{attribute 'no_explicit_call':= 'do not call this POU directly'}
FUNCTION_BLOCK TValueMonitor
VAR
    _CurrentValue : INT := -1;
    _PreviousValue : INT;
    _Changed : BOOL;
END_VAR

PROPERTY Changed : BOOL
GET
Changed := _Changed;
END_GET
END_PROPERTY

PROPERTY CurrentValue : INT
GET
CurrentValue := _CurrentValue;
END_GET
END_PROPERTY

PROPERTY PreviousValue : INT
GET
PreviousValue := _PreviousValue;
END_GET
END_PROPERTY

METHOD Reset
VAR_INPUT
END_VAR
_CurrentValue := 0;
_PreviousValue := 0;
END_METHOD

METHOD Test : BOOL
VAR_INPUT
    Value : INT;
END_VAR
_Changed := Value <> _CurrentValue;
_PreviousValue := _CurrentValue;
_CurrentValue := Value;

Test := _Changed;
END_METHOD

END_FUNCTION_BLOCK

(* stored: Version 1.1.0.1, ProductVersion 3.1.4024.3
   POU TValueMonitor: Id {83feb238-a6d0-08e1-3d2f-4edc7cda39f9}, SpecialFunc None
   Property Changed: Id {64ce711e-c886-01bc-2998-59a84e0dabaa}
   Get Get: Id {d78bc9d3-e9b4-02d1-10c2-43392bf24118}
   Property CurrentValue: Id {08c4126c-4fb0-030a-15b8-ed065e961df7}
   Get Get: Id {03b0f48f-50fc-0a77-28db-25f1a3089478}
   Property PreviousValue: Id {d5cb63eb-1062-0765-07ce-1c857312fc00}
   Get Get: Id {045dbc11-1e3f-0f62-2567-30f4a71eb43d}
   Method Reset: Id {0448d132-9779-0606-12cd-041f8768b4e1}
   Method Test: Id {3611567e-1683-0480-2672-5b7b7e8ea200} *)
